// Mitsubishi GX Works2 project: e02   PLC: Q02/Q02H

PROGRAM MAIN
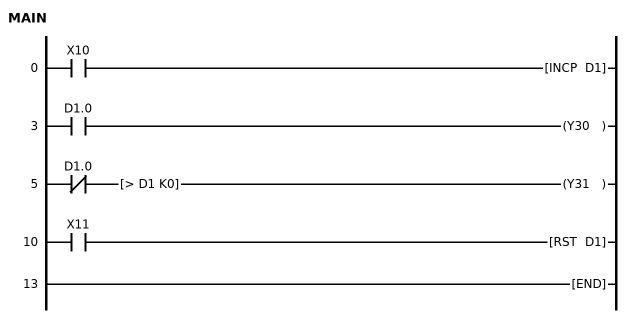
0     LD      X10
      INCP    D1
3     LD      D1.0
      OUT     Y30
5     LDI     D1.0
      AND>    D1 K0
      OUT     Y31
10    LD      X11
      RST     D1
13    END
END_PROGRAM
